Staubli VAL3: goTo.pgx

program goTo(num x_nIndex, bool& x_bUnreached[])
  local bool l_bUnreached
  local num l_nIndexTool
  local tool l_tTool
begin
end
